{attribute addProperty BoxType "EL3052-0000-0017"}
{attribute addProperty Id "AI_Standard_ChannelAT %I*ARRAY[0..2] OF AI_Standard_Channel_B51B79FC16220.250WcStateAT %I*WcState_98A4DF7520.250InfoDataAT %I*InfoData_BC63D37F80100"}
{attribute addProperty CRC "2847295426"}
{attribute addProperty SizeInBites "244"}
{attribute addProperty SizeInBytes "30.5"}
TYPE EL3052_4AB1F135 :
STRUCT
	{attribute addProperty Name "AI_Standard_Channel"}
	AI_Standard_Channel : ARRAY[0..2] OF AI_Standard_Channel_B51B79FC;
	{attribute addProperty Name "WcState"}
	WcState : WcState_98A4DF75;
	{attribute addProperty Name "InfoData"}
	InfoData : InfoData_BC63D37F;
END_STRUCT
END_TYPE

(* stored: Version 1.2.0.0, ProductVersion 3.1.4024.9
   DUT EL3052_4AB1F135: Id {c2884d25-51de-4dba-8123-915dccb29903} *)
